DATA_BLOCK "PartDataManage_Part1_DB"
{ S7_Optimized_Access := 'TRUE' }
VERSION : 0.1
NON_RETAIN
// ATTRIBUTES
// AUTO_NUMBER = True
// BLOCK_NUMBER = 1501
// END_ATTRIBUTES
"PartDataManage"

BEGIN

END_DATA_BLOCK

